Staubli VAL3: stringinit.pgx

program stringinit()
  local num i
  local string l_str
begin
  //  for i=0 to 500
  //    $dins(sTxtfile,i)
  //    l_str=toString("1",i)
  //    sTxtfile[i]="path"+l_str+".txt"
  //  endFor
end
